SUBAPPLICATION Counter (* Subapplication Type *)
  (* Standard: 61499-2 *)
  (* Version 1.0, 2023-02-17, Franz *)
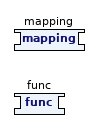
  SUBAPPS
    mapping : mapping;
    func : func;
  END_SUBAPPS
END_SUBAPPLICATION
